{attribute 'Tc2GvlVarNames'}
VAR_GLOBAL
	Palp_R						: ARRAY[1..3] OF Points_Palpage_Laser;	(* Face1 : Aile Ref ; Face2 : Ame ; Face3 : Aile Opp Ref *)
	M, Angles_Rotation			: ARRAY[1..3] OF Coordonnees;			(* Face1 : Aile Ref ; Face2 : Ame ; Face3 : Aile Opp Ref *)
	limite_couple_negatif_axe_Z_Laser	AT%Q*:INT;
END_VAR

(* stored: Version 1.1.0.1, ProductVersion 3.1.4024.15
   GVL Palpage_laser: Id {a40d9036-2c23-4faf-8149-ee8806c0003f} *)
